Fanuc KAREL source: kt00857.KL

-- PROVISIONAL review KL for V940-1; original PC SHA256 5d9ee332d1943f31f0e408633dccdbc6b6593504c6ecefbc2a73f9020356d741
-- Incomplete behavior may be omitted. Consult companion uncertainty JSON. Do not deploy.
PROGRAM KT00857
%NOLOCKGROUP
VAR
  I1 : INTEGER
  I2 : INTEGER
  OUT : REAL
BEGIN
  -- V9_ZERO_TABLE_METADATA_HINT layout=0001; no indexed target words; source/name/runtime held
  -- UNRESOLVED_PC offsets 5-16; opcodes 2E,23
  -- UNRESOLVED_PC offsets 21-32; opcodes 2E,23
  -- UNRESOLVED_PC offsets 37-48; opcodes 2E,23
  -- UNRESOLVED_PC offsets 53-64; opcodes 2E,23
  -- UNRESOLVED_PC offsets 69-87; opcodes 27,27,21,64,76,64,23
  -- UNRESOLVED_PC offsets 92-96; opcodes 7F
END KT00857
